# B&R Automation Studio project ST
Automation Studio 4.9

## Configuration Config1

CPU X20CP1584, AutomationRuntime B4.93, Build 4.1.2, Vc V4.72.6

### Task classes (Cpu.sw)
```
Cyclic#4:
  Cosberg <- Cosberg.prg
```

### Hardware
```
X20CP1584 : X20CP1584 v1.10.0.0
  Connector IF2:
    ActivateDevice = 1
  ConfigurationID = ST_Config1
  Simulation = 1
  FileDevice1
  FileDeviceName1 = USER
  FileDevicePath1 = USER_PATH
```

## Logical view

### Program Logical/Cosberg (IEC)

#### Cyclic.st - Cyclic code
```iecst
PROGRAM _CYCLIC

	CASE STATO OF
		STATO_SPENTO: // attendiamo l'avvio
			// attivazione del nastro trasportatore
			IF NASTRO_ON THEN
				STATO := STATO_ACCESO;
				NASTRO_ON:= FALSE;
			END_IF;

		STATO_ACCESO:

			// In caso di emergenza spegnamo tutto senza pensarci due volte e cambiamo stato
			IF STOP_EMERGENZA THEN
				ALIMENTAZIONE := 0;
				SALDATURA_ON := 0;
				FORATURA_ON := 0;
				AVVITATURA_ON := 0;
				QUALITY_CHECK := 0;
				// cambiamo stato
				STATO := STATO_SPENTO;
			ELSE  // se non c'è emergenza lavoriamo normalmente
				// se è presente un pezzo in staz_1
				IF STAZ_1 AND C_MAN_IN < CILCI_MANUTENZIONE THEN
					// chiamo la funzione per la stazione 1
					GESTIONE_STAZ_1(TIPO := TIPO_TRIGGER , TEMPO :=  T#0s , TRIGGER :=  PRESENZA_PEZZO, AZIONE := ALIMENTAZIONE);
					// se si verifica l'edge negativo disattivo la stazione e conto il pezzo
					IF EDGENEG(ALIMENTAZIONE) THEN
						PRESENZA_PEZZO := FALSE;
						STAZ_1 := FALSE;
						C_MAN_IN := C_MAN_IN + 1;
					END_IF;
				END_IF;
				// se è presente un pezzo in staz_2
				IF STAZ_2 THEN
					// chiamo la funzione per la stazione 2
					GESTIONE_STAZ_2(TIPO := TIPO_TEMPO , TEMPO :=  T#5s , TRIGGER :=  FALSE , AZIONE := SALDATURA_ON);
					// se si verifica l'edge negativo disattivo la stazione
					STAZ_2 := NOT EDGENEG(SALDATURA_ON);
				END_IF;
				// se è presente un pezzo in staz_3
				IF STAZ_3 THEN
					// chiamo la funzione per la stazione 3
					GESTIONE_STAZ_3(TIPO := TIPO_TEMPO , TEMPO :=  T#3s , TRIGGER := FALSE, AZIONE := FORATURA_ON);
					// se si verifica l'edge negativo disattivo la stazione
					STAZ_3 := NOT EDGENEG(FORATURA_ON);
				END_IF;
				// se è presente un pezzo in staz_4
				IF STAZ_4 THEN
					// chiamo la funzione per la stazione 4
					GESTIONE_STAZ_4(TIPO := TIPO_TEMPO , TEMPO :=  T#4s , TRIGGER :=  FALSE, AZIONE := AVVITATURA_ON);
					// se si verifica l'edge negativo disattivo la stazione
					STAZ_4 := NOT EDGENEG(AVVITATURA_ON);
				END_IF;
				// se è presente un pezzo in staz_5
				IF STAZ_5 THEN
					// chiamo la funzione per la stazione 5
					GESTIONE_STAZ_5(TIPO := TIPO_TRIGGER , TEMPO :=  T#0s , TRIGGER :=  QUALITY_CHECK_DONE, AZIONE := QUALITY_CHECK);
					// se si verifica l'edge negativo disattivo la stazione e incremento il contatore finale
					IF EDGENEG(QUALITY_CHECK) THEN
						QUALITY_CHECK_DONE := FALSE;
						STAZ_5 := FALSE;
						C_MAN_OUT := C_MAN_OUT + 1;
					END_IF;
				END_IF;
				// verifichiamo se l'ultimo pezzo è uscito dalla stazione
				IF C_MAN_OUT >= CILCI_MANUTENZIONE THEN
						STATO := STATO_MANUTENZIONE;
				END_IF;
			END_IF;

		STATO_MANUTENZIONE:
			MAI := TRUE;
			IF MAIR THEN
				C_MAN_IN := 0;
				C_MAN_OUT := 0;
				MAI := FALSE;
				MAIR := FALSE;
				STATO := STATO_ACCESO;

			END_IF;
	END_CASE;
END_PROGRAM
```

#### Variables.var - Local variables
```iecst
VAR CONSTANT
	TIPO_TRIGGER : USINT := 0;
	TIPO_TEMPO : USINT := 1;
END_VAR
VAR
	STOP_EMERGENZA : BOOL;
	STAZ_5 : BOOL;
	STAZ_4 : BOOL;
	STAZ_3 : BOOL;
	STAZ_2 : BOOL;
	STAZ_1 : BOOL;
END_VAR
VAR CONSTANT
	STATO_SPENTO : USINT := 0;
	STATO_MANUTENZIONE : USINT := 2;
	STATO_ACCESO : USINT := 1;
END_VAR
VAR
	STATO : {REDUND_UNREPLICABLE} USINT := 0;
	SALDATURA_ON : BOOL;
	QUALITY_CHECK_DONE : BOOL;
	QUALITY_CHECK : BOOL;
	PRESENZA_PEZZO : BOOL;
	NASTRO_ON : BOOL;
	MAIR : BOOL;
	MAI : BOOL;
	GESTIONE_STAZ_5 : GESTIONE_STAZIONE;
	GESTIONE_STAZ_4 : GESTIONE_STAZIONE;
	GESTIONE_STAZ_3 : GESTIONE_STAZIONE;
	GESTIONE_STAZ_2 : GESTIONE_STAZIONE;
	GESTIONE_STAZ_1 : GESTIONE_STAZIONE;
	FORATURA_ON : BOOL;
	C_MAN_OUT : USINT;
	C_MAN_IN : USINT;
	CILCI_MANUTENZIONE : {REDUND_UNREPLICABLE} USINT := 10;
	AVVITATURA_ON : BOOL;
	ALIMENTAZIONE : BOOL;
END_VAR
```

#### LocalFunctions.fun
```iecst
{REDUND_ERROR} FUNCTION_BLOCK GESTIONE_STAZIONE (*TODO: Add your comment here*) (*$GROUP=User,$CAT=User,$GROUPICON=User.png,$CATICON=User.png*)
	VAR_INPUT
		TIPO : USINT;
		TEMPO : TIME;
		TRIGGER : BOOL;
	END_VAR
	VAR_IN_OUT
		AZIONE : BOOL;
	END_VAR
	VAR
		TEMPORIZZATORE : TIME := T#0s;
	END_VAR
	VAR CONSTANT
		TIPO_TRIGGER : USINT := 0;
		TIPO_TEMPO : USINT := 1;
	END_VAR
	VAR
		EVENTO : BOOL;
		zzEdge00000 : BOOL;
	END_VAR
	VAR CONSTANT
		DELTA_T : TIME := T#100ms;
	END_VAR
END_FUNCTION_BLOCK
```

#### GESTIONE_STAZIONE.st
```iecst
(* function block per la gestione delle singole stazioni *)
FUNCTION_BLOCK GESTIONE_STAZIONE

	AZIONE:= TRUE;

	CASE TIPO OF
		TIPO_TRIGGER:
			// se è presente il fornte positivo di trigger
			IF EDGEPOS(TRIGGER) THEN
				// segnalo che è avvenuto l'evento
				EVENTO:= TRUE;
			END_IF;

		TIPO_TEMPO:
			//incremento del temporizzatore
			TEMPORIZZATORE := TEMPORIZZATORE + DELTA_T;
			// verifica superamento del tempo
			IF TEMPORIZZATORE >= TEMPO THEN
				EVENTO:= TRUE;
			END_IF;
	END_CASE;

	// gestione azioni se si verifica l'evento
	IF EVENTO THEN
		AZIONE:= FALSE;
		TEMPORIZZATORE:= T#0s;
		TRIGGER:= FALSE;
		EVENTO := FALSE;
	END_IF;

END_FUNCTION_BLOCK
```

Listed in the project but not available here: Logical/Global.typ, Logical/Global.var, Logical/Libraries, Logical/Cosberg/Init.st, Logical/Cosberg/Exit.st, Logical/Cosberg/Types.typ
